(* Logix 5000 project; controller Chia_Dynamix_Seguridad Emulate 5570 rev 30.12; software revision 30.00 *)

TASK T00_MainTask (continuous, watchdog 500 ms) : M00_MainProgram

MODULES
   Local : Emulate 5570 (ICP 6, rev 30.12)
      Salidas_Digitales : vendor 1 type 7 code 16 (ICP 4, rev 3.1, Output RPI 20 ms)
      PLC1 : Emulate 5570 (ICP 2, rev 30.1, $b0c4f640$ RPI 20 ms, $2aa0071a$ RPI 20 ms, $47fd6544$ RPI 20 ms, $78934f3e$ RPI 20 ms, $e7fd9788$ RPI 20 ms, $e4a915d0$ RPI 20 ms, $e3153c45$ RPI 20 ms, $817deb3b$ RPI 20 ms)
      PlC2 : Emulate 5570 (ICP 5, rev 30.1, $a46f44a2$ RPI 20 ms, $a059310c$ RPI 20 ms, $2bedab46$ RPI 20 ms, $e229f641$ RPI 20 ms, $a5fb9b3a$ RPI 20 ms, $1ba65c8b$ RPI 20 ms, $d241e22c$ RPI 20 ms, $a9cd2d66$ RPI 20 ms)
END_MODULES

VAR_GLOBAL   (* controller tags *)
   BALIZA_SEGURIDAD_AMARILLO : ALIAS FOR Local:4:I.Data.0;   // Indica operación de Mantenimiento activa
   BALIZA_SEGURIDAD_EMERGENCIA : ALIAS FOR Local:4:I.Data.1;   // Prende-Apaga: Indica que algún elemento de seguridad ha sido activado
   BALIZA_SEGURIDAD_ROJO : ALIAS FOR Local:4:I.Data.2;   // Continua: Indica que el botón de parada se encuentra activo
   BALIZA_SEGURIDAD_VERDE : ALIAS FOR Local:4:I.Data.3;   // Indica Procedimiento Automático Normal, sin errores
   Controles_Permisivos : DINT; {produced}   // Señal que al estar activa indica que algun elemento de seguridad ha sido activado
   FAB_CER_AUTO_BTN : DINT;   // Botón de Inicio Automático
   FAB_CER_EME_BTN1 : DINT := 1;   // Botón de Emergencia NO, se recibe del PLC1
   FAB_CER_EME_BTN2 : DINT := 1;   // Botón de Emergencia NA, se recibe del PLC2
   FAB_CER_HOMBRE_MUERTO : DINT := 1;   // Botón de emergencia ligado a la rutina de robot NC
   FAB_CER_RESET1 : DINT;   // Botón de Reset del PLC1
   FAB_CER_RESET2 : DINT;   // Botón de Reset del PLC2
   FAB_CER_SCANNER_AREA : DINT := 1;   // Señal NC que indica si hay alguna presencia no autorizada.
   FAB_CER_STP1 : DINT;   // Botón de Parada del PLC1
   FAB_CER_STP2 : DINT;   // Botón de Parada del PLC2
   FAB_CER_STT_BTN : DINT;   // Botón de Start
   FAB_CER_TAPETE_SEGURIDAD : DINT := 1;   // Señal NC que indica si hay alguna presencia no autorizada.
   FAB_CORTINAS_SEGURIDAD1 : DINT := 1;   // Señal NC que indica si las cortina1 de seguridad han sido interrumpidas
   FAB_CORTINAS_SEGURIDAD2 : DINT := 1;   // Señal NC que indica si las cortina2 de seguridad han sido interrumpidas
   FAB_INTERLOCK_PUERTA1 : DINT := 1;   // Señal NC que indica si la puerta de la celda robótica se encuentra abierta
   FAB_INTERLOCK_PUERTA2 : DINT := 1;   // Señal NC que indica si la puerta de la celda robótica se encuentra abierta
   SIGNAL_MAINT : DINT;   // Señal que indica que se están realizando operaciones de mantenimiento
   SIGNAL_RESET : BOOL;   // Señal que indica que algún Botón de Reset ha sido presionado
   SIGNAL_TIMER : BOOL;   // Señal que indica que los 3 segundos del botón automático se han completado
   TIMER_START : TIMER := (PRE := 3000);   // Timer que lleva el conteo de 3 segundos para habilitar el modo automático
END_VAR

PROGRAM M00_MainProgram   (* main routine R00_MainRoutine *)

ROUTINE R00_MainRoutine   (* ladder *)
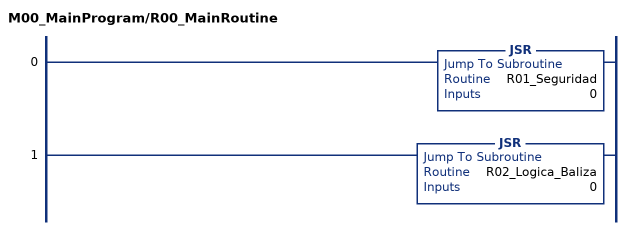
   0: JSR(R01_Seguridad,0);
   1: JSR(R02_Logica_Baliza,0);
END_ROUTINE

ROUTINE R01_Seguridad   (* ladder *)
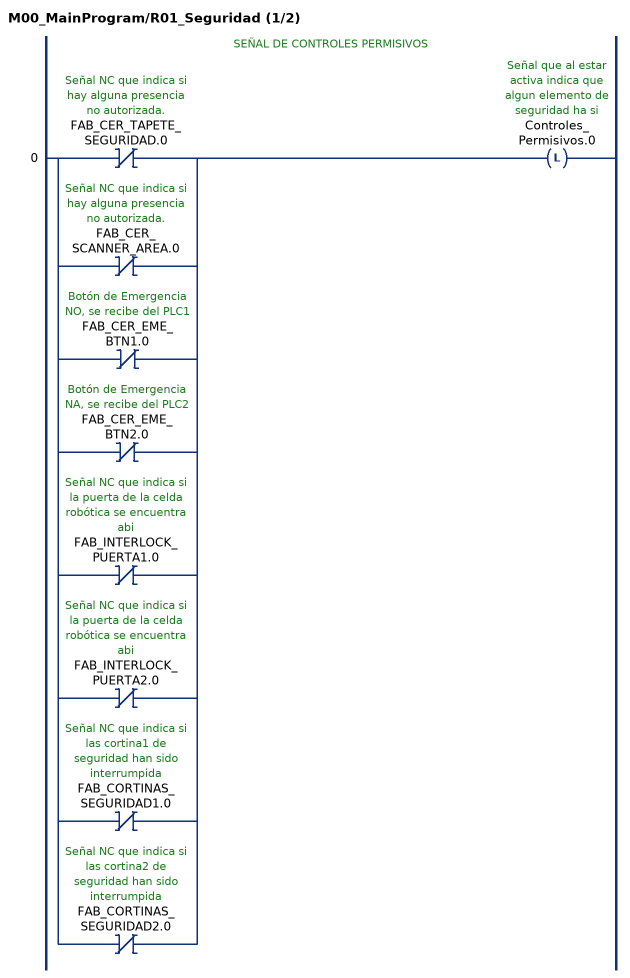
   // SEÑAL DE CONTROLES PERMISIVOS
   0: [XIO(FAB_CER_TAPETE_SEGURIDAD.0) ,XIO(FAB_CER_SCANNER_AREA.0) ,XIO(FAB_CER_EME_BTN1.0) ,XIO(FAB_CER_EME_BTN2.0) ,XIO(FAB_INTERLOCK_PUERTA1.0) ,XIO(FAB_INTERLOCK_PUERTA2.0) ,XIO(FAB_CORTINAS_SEGURIDAD1.0) ,XIO(FAB_CORTINAS_SEGURIDAD2.0) ]OTL(Controles_Permisivos.0);
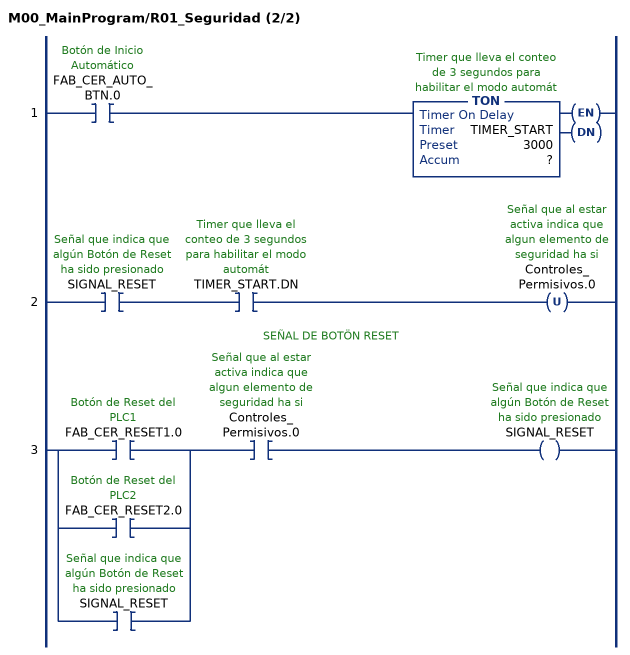
   1: XIC(FAB_CER_AUTO_BTN.0)TON(TIMER_START,?,?);
   2: XIC(SIGNAL_RESET)XIC(TIMER_START.DN)OTU(Controles_Permisivos.0);
   // SEÑAL DE BOTÖN RESET
   3: [XIC(FAB_CER_RESET1.0) ,XIC(FAB_CER_RESET2.0) ,XIC(SIGNAL_RESET) ]XIC(Controles_Permisivos.0)OTE(SIGNAL_RESET);
END_ROUTINE

ROUTINE R02_Logica_Baliza   (* ladder *)
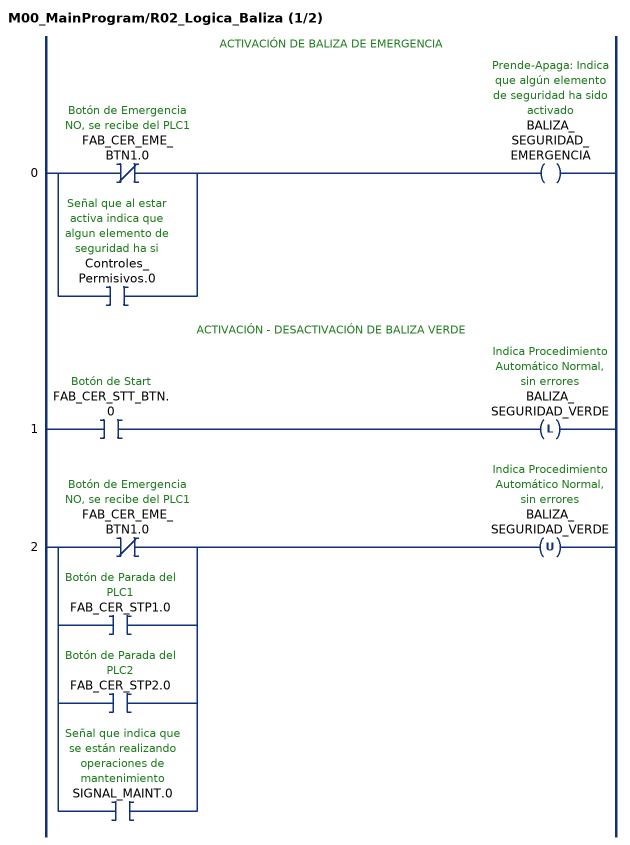
   // ACTIVACIÓN DE BALIZA DE EMERGENCIA
   0: [XIO(FAB_CER_EME_BTN1.0) ,XIC(Controles_Permisivos.0) ]OTE(BALIZA_SEGURIDAD_EMERGENCIA);
   // ACTIVACIÓN - DESACTIVACIÓN DE BALIZA VERDE
   1: XIC(FAB_CER_STT_BTN.0)OTL(BALIZA_SEGURIDAD_VERDE);
   2: [XIO(FAB_CER_EME_BTN1.0) ,XIC(FAB_CER_STP1.0) ,XIC(FAB_CER_STP2.0) ,XIC(SIGNAL_MAINT.0) ]OTU(BALIZA_SEGURIDAD_VERDE);
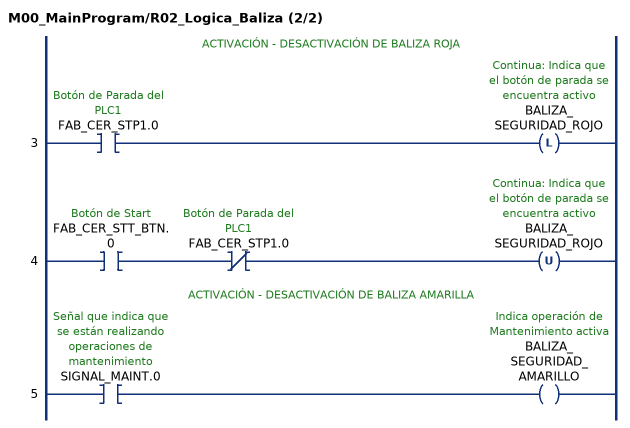
   // ACTIVACIÓN - DESACTIVACIÓN DE BALIZA ROJA
   3: XIC(FAB_CER_STP1.0)OTL(BALIZA_SEGURIDAD_ROJO);
   4: XIC(FAB_CER_STT_BTN.0)XIO(FAB_CER_STP1.0)OTU(BALIZA_SEGURIDAD_ROJO);
   // ACTIVACIÓN - DESACTIVACIÓN DE BALIZA AMARILLA
   5: XIC(SIGNAL_MAINT.0)OTE(BALIZA_SEGURIDAD_AMARILLO);
END_ROUTINE
END_PROGRAM
